Staubli VAL3: atiForceSen7.pjx

--- atiForceSen7.pjx ---
Parameters version=s7.3.1 stackSize=5000 millimeterUnit=true
Program file=initialize.pgx
Program file=loopReadForce.pgx
Program file=readForce.pgx
Program file=readme.pgx
Program file=start.pgx
Program file=stop.pgx
Program file=user.pgx
Data file=atiForceSen7.dtx

--- atiForceSen7.dtx ---
bool bClear
bool bOverRun
public bool bZero
mdesc mNomSpeed
public num nForce[6]
num nHeader[2]
num nMonitor[2]
num nPort = 49151
num nRec[16]
num nReceived = -1
num nScaleForce = 6104
num nScaleTorque = 153
num nSend[20]
num nSent = -1
num nSioTimeOut = 5
public num nStatus
num nVecForce
sio sFs = {link=Socket\sAtiFs}
num nCountPerFs
num nCountPerTq

--- start.pgx ---
program start()
  local num l_n
begin
  //Header begin
  //Description of Program
  // ATI Force Sensor
  // run as test of sensor
  // or use applicaiton as library
  //
  //Input parameters
  // none
  //
  //Output parameters
  // none
  //
  //Examples
  // run
  //
  //History
  // Creation: 10-Jul-2009, J Cook
  // Modification: 28-Feb-2013, yeyonglong
  //  description continued
  //
  //Header end
  call initialize("io:sAtiFs",l_n)
  taskCreateSync "readForce",0.01,bOverRun,loopReadForce()
  taskCreate "user",100,user()
end

--- readForce.pgx ---
program readForce(num& x_nStatus, num& x_nForce[], num& x_nMonitor[], bool& x_bZero, bool& x_bClear)
  local num l_n
begin
  //Header begin
  //Description of Program
  // Reads ATI Force Sensor values
  // Usually ran in a synchronous task
  //
  //Input parameters
  // none
  //
  //Output parameters
  // num    x_nStatus : Returns status of sensor
  // num    x_nForce  : Array of 6 num that returns force and moment values
  // num    x_nMonitor: Array of 2 num that sets monitor bits
  // bool   x_bZero   : Set to zero (tare) sensor, reset when request is sent
  // bool   x_bClear  ; set to clear monitor conditions, reset when reguest is sent
  //
  //Examples
  // taskCreateSync "readForce",0.004,bOverRun,readForce(nStatus,nForce,nMonitor,bZero,bClear)
  //
  //History
  // Creation: 10-Jul-2009, J Cook
  // Modification: 28-Feb-2013, yeyonglong, update to v7
  // description continued
  //
  //Header end
  nSend[16]=round(limit(x_nMonitor[1],0,255))
  nSend[17]=round(limit(x_nMonitor[0],0,255))
  if x_bZero==true
    nSend[19]=bOr(nSend[19],1)
  endIf
  if x_bClear==true
    nSend[19]=bOr(nSend[19],2)
  endIf
  nSent=sioSet(sFs,nSend)
  if nSent!=size(nSend)
    x_nStatus=-1
  else
    nSend[19]=0
  endIf
  nReceived=sioGet(sFs,nRec)
  if nReceived!=16
    x_nStatus=-2
  endIf
  if nRec[0]==nHeader[0] and nRec[1]==nHeader[1]
    x_nStatus=(nRec[3]+nRec[2]*256)
    for l_n=0 to 5
      x_nForce[l_n]=(nRec[(l_n*2)+5]+nRec[(l_n*2)+4]*256)
      if x_nForce[l_n]>power(2,15)
        x_nForce[l_n]=x_nForce[l_n]-power(2,16)
      endIf
      if l_n<=2
        x_nForce[l_n]=x_nForce[l_n]/nCountPerFs*nScaleForce
      else
        x_nForce[l_n]=x_nForce[l_n]/nCountPerTq*nScaleTorque
      endIf
    endFor
  else
    x_nStatus=-3
  endIf
  nVecForce=sqrt(x_nForce[0]*x_nForce[0]+x_nForce[1]*x_nForce[1]+x_nForce[2]*x_nForce[2])
end

--- readme.pgx ---
program readme()
begin
  //TITLE             : ATI force sensor
  //General desription: reads values from ATI force sensor with TCP/IP Socket interface
  //Hardware Required : ATI Force Sensor
  //Library Version   : 7.3.1
  //Public Variables  : bZero nForce nStatus
  //Public Program    : initialize() loopReadForce()
  //Included Libraries: None
  //Miscellaneous     : Requires a TCP/IP Client socket
  //Keywords          : ATI Force Sensor
end

--- user.pgx ---
program user()
  local num l_nKey
begin
  //Header begin
  //Description of Program
  // Output page for test
  //
  //Input parameters
  // none
  //
  //Output parameters
  // none
  //
  //Examples
  // taskCreate "user",100,user()
  //
  //History
  // Creation: 10-Jul-2009, J Cook
  // Modification: 28-Feb-2013, yeyonglong
  //  description continued
  //
  //Header end
  userPage()
  do
    cls()
    put("status: ")
    putln(nStatus)
    put("fX: ")
    putln(nForce[0])
    put("fY: ")
    putln(nForce[1])
    put("fZ: ")
    putln(nForce[2])
    put("mX: ")
    putln(nForce[3])
    put("mY: ")
    putln(nForce[4])
    put("mZ: ")
    putln(nForce[5])
    gotoxy(0,9)
    put("Force Vec: ")
    put(nVecForce)
    gotoxy(0,13)
    put("ZERO")
    l_nKey=getKey()
    switch l_nKey
      case 271
        bZero=true
      break
    endSwitch
    delay(0)
  until false
end
